// EAP paras
// Additional Services
EAP_paras^.AdditonalSerivce.Reserved1 := DINT_TO_REAL(EAP_para_DINT^.AdditonalSerivce.Reserved1);
EAP_paras^.AdditonalSerivce.Reserved2 := DINT_TO_REAL(EAP_para_DINT^.AdditonalSerivce.Reserved2);
EAP_paras^.AdditonalSerivce.Reserved3 := DINT_TO_REAL(EAP_para_DINT^.AdditonalSerivce.Reserved3);
EAP_paras^.AdditonalSerivce.Reserved4 := DINT_TO_REAL(EAP_para_DINT^.AdditonalSerivce.Reserved4);
EAP_paras^.AdditonalSerivce.Reserved5 := DINT_TO_REAL(EAP_para_DINT^.AdditonalSerivce.Reserved5);
EAP_paras^.AdditonalSerivce.Reserved6 := DINT_TO_REAL(EAP_para_DINT^.AdditonalSerivce.Reserved6);
EAP_paras^.AdditonalSerivce.Reserved7 := DINT_TO_REAL(EAP_para_DINT^.AdditonalSerivce.Reserved7);
EAP_paras^.AdditonalSerivce.Reserved8 := DINT_TO_REAL(EAP_para_DINT^.AdditonalSerivce.Reserved8);
EAP_paras^.AdditonalSerivce.Reserved9 := DINT_TO_REAL(EAP_para_DINT^.AdditonalSerivce.Reserved9);
EAP_paras^.AdditonalSerivce.Reserved10 := DINT_TO_REAL(EAP_para_DINT^.AdditonalSerivce.Reserved10);
EAP_paras^.AdditonalSerivce.Reserved11 := DINT_TO_REAL(EAP_para_DINT^.AdditonalSerivce.Reserved11);
EAP_paras^.AdditonalSerivce.Reserved12 := DINT_TO_REAL(EAP_para_DINT^.AdditonalSerivce.Reserved12);
EAP_paras^.AdditonalSerivce.Reserved13 := DINT_TO_REAL(EAP_para_DINT^.AdditonalSerivce.Reserved13);
EAP_paras^.AdditonalSerivce.Reserved14 := DINT_TO_REAL(EAP_para_DINT^.AdditonalSerivce.Reserved14);
EAP_paras^.AdditonalSerivce.Reserved15 := DINT_TO_REAL(EAP_para_DINT^.AdditonalSerivce.Reserved15);
EAP_paras^.AdditonalSerivce.Reserved16 := DINT_TO_REAL(EAP_para_DINT^.AdditonalSerivce.Reserved16);
//CommonBlock_Params
EAP_paras^.CommonBlock_Params_EAP.ActivePowerLimit := DINT_TO_REAL(EAP_para_DINT^.CommonBlock_Params_EAP.ActivePowerLimit);
EAP_paras^.CommonBlock_Params_EAP.Delta_limits := DINT_TO_REAL(EAP_para_DINT^.CommonBlock_Params_EAP.Delta_limits);
EAP_paras^.CommonBlock_Params_EAP.E_Limits := DINT_TO_REAL(EAP_para_DINT^.CommonBlock_Params_EAP.E_Limits)*0.1;
EAP_paras^.CommonBlock_Params_EAP.Ki_ReactiveControl := DINT_TO_REAL(EAP_para_DINT^.CommonBlock_Params_EAP.Ki_ReactiveControl)*0.0001;
EAP_paras^.CommonBlock_Params_EAP.Kp_ReactiveControl := DINT_TO_REAL(EAP_para_DINT^.CommonBlock_Params_EAP.Kp_ReactiveControl)*0.0001;
EAP_paras^.CommonBlock_Params_EAP.NominalFreq := DINT_TO_REAL(EAP_para_DINT^.CommonBlock_Params_EAP.NominalFreq);
EAP_paras^.CommonBlock_Params_EAP.NominalPower := DINT_TO_REAL(EAP_para_DINT^.CommonBlock_Params_EAP.NominalPower);
EAP_paras^.CommonBlock_Params_EAP.NominalVolt := DINT_TO_REAL(EAP_para_DINT^.CommonBlock_Params_EAP.NominalVolt);
EAP_paras^.CommonBlock_Params_EAP.ReactivePowerLimit := DINT_TO_REAL(EAP_para_DINT^.CommonBlock_Params_EAP.ReactivePowerLimit);
EAP_paras^.CommonBlock_Params_EAP.VirtualReactance := DINT_TO_REAL(EAP_para_DINT^.CommonBlock_Params_EAP.VirtualReactance)*0.001;
EAP_paras^.CommonBlock_Params_EAP.VirtualResistor := DINT_TO_REAL(EAP_para_DINT^.CommonBlock_Params_EAP.VirtualResistor)*0.001;
EAP_paras^.CommonBlock_Params_EAP.Reserved1 := DINT_TO_REAL(EAP_para_DINT^.CommonBlock_Params_EAP.Reserved1);
EAP_paras^.CommonBlock_Params_EAP.Reserved2 := DINT_TO_REAL(EAP_para_DINT^.CommonBlock_Params_EAP.Reserved2);
EAP_paras^.CommonBlock_Params_EAP.Reserved3 := DINT_TO_REAL(EAP_para_DINT^.CommonBlock_Params_EAP.Reserved3);
EAP_paras^.CommonBlock_Params_EAP.Reserved4 := DINT_TO_REAL(EAP_para_DINT^.CommonBlock_Params_EAP.Reserved4);
EAP_paras^.CommonBlock_Params_EAP.Reserved5 := DINT_TO_REAL(EAP_para_DINT^.CommonBlock_Params_EAP.Reserved5);
//FrequencyRegulation_Params
EAP_paras^.FrequencyRegulation_Params_EAP.DeadBand_Limits_P := DINT_TO_REAL(EAP_para_DINT^.FrequencyRegulation_Params_EAP.DeadBand_Limits_P)*0.1;
EAP_paras^.FrequencyRegulation_Params_EAP.DroopConstantP := DINT_TO_REAL(EAP_para_DINT^.FrequencyRegulation_Params_EAP.DroopConstantP)*0.1;
EAP_paras^.FrequencyRegulation_Params_EAP.LowPassFilter_CutOff_Freq := DINT_TO_REAL(EAP_para_DINT^.FrequencyRegulation_Params_EAP.LowPassFilter_CutOff_Freq)*0.01;
EAP_paras^.FrequencyRegulation_Params_EAP.Max_Delta_Energy := DINT_TO_REAL(EAP_para_DINT^.FrequencyRegulation_Params_EAP.Max_Delta_Energy);
EAP_paras^.FrequencyRegulation_Params_EAP.PowerLimit_Freq := DINT_TO_REAL(EAP_para_DINT^.FrequencyRegulation_Params_EAP.PowerLimit_Freq);
EAP_paras^.FrequencyRegulation_Params_EAP.Reserved1 := DINT_TO_REAL(EAP_para_DINT^.FrequencyRegulation_Params_EAP.Reserved1);
EAP_paras^.FrequencyRegulation_Params_EAP.Reserved2 := DINT_TO_REAL(EAP_para_DINT^.FrequencyRegulation_Params_EAP.Reserved2);
EAP_paras^.FrequencyRegulation_Params_EAP.Reserved3 := DINT_TO_REAL(EAP_para_DINT^.FrequencyRegulation_Params_EAP.Reserved3);
EAP_paras^.FrequencyRegulation_Params_EAP.Reserved4 := DINT_TO_REAL(EAP_para_DINT^.FrequencyRegulation_Params_EAP.Reserved4);
EAP_paras^.FrequencyRegulation_Params_EAP.Reserved5 := DINT_TO_REAL(EAP_para_DINT^.FrequencyRegulation_Params_EAP.Reserved5);
EAP_paras^.FrequencyRegulation_Params_EAP.Reserved6 := DINT_TO_REAL(EAP_para_DINT^.FrequencyRegulation_Params_EAP.Reserved6);
EAP_paras^.FrequencyRegulation_Params_EAP.Reserved7 := DINT_TO_REAL(EAP_para_DINT^.FrequencyRegulation_Params_EAP.Reserved7);
EAP_paras^.FrequencyRegulation_Params_EAP.Reserved8 := DINT_TO_REAL(EAP_para_DINT^.FrequencyRegulation_Params_EAP.Reserved8);
EAP_paras^.FrequencyRegulation_Params_EAP.Reserved9 := DINT_TO_REAL(EAP_para_DINT^.FrequencyRegulation_Params_EAP.Reserved9);
EAP_paras^.FrequencyRegulation_Params_EAP.Reserved10 := DINT_TO_REAL(EAP_para_DINT^.FrequencyRegulation_Params_EAP.Reserved10);
EAP_paras^.FrequencyRegulation_Params_EAP.Reserved11 := DINT_TO_REAL(EAP_para_DINT^.FrequencyRegulation_Params_EAP.Reserved11);
//InertiaEmulation_Params
EAP_paras^.InertiaEmulation_Params_EAP.Damping_Constant := DINT_TO_REAL(EAP_para_DINT^.InertiaEmulation_Params_EAP.Damping_Constant)*0.1;
EAP_paras^.InertiaEmulation_Params_EAP.HighPassFilterConst := DINT_TO_REAL(EAP_para_DINT^.InertiaEmulation_Params_EAP.HighPassFilterConst)*0.001;
EAP_paras^.InertiaEmulation_Params_EAP.Inertia_Constant := DINT_TO_REAL(EAP_para_DINT^.InertiaEmulation_Params_EAP.Inertia_Constant)*0.1;
EAP_paras^.InertiaEmulation_Params_EAP.Max_ROCOF := DINT_TO_REAL(EAP_para_DINT^.InertiaEmulation_Params_EAP.Max_ROCOF)*0.01;
EAP_paras^.InertiaEmulation_Params_EAP.Reserved1 := DINT_TO_REAL(EAP_para_DINT^.InertiaEmulation_Params_EAP.Reserved1);
EAP_paras^.InertiaEmulation_Params_EAP.Reserved2 := DINT_TO_REAL(EAP_para_DINT^.InertiaEmulation_Params_EAP.Reserved2);
EAP_paras^.InertiaEmulation_Params_EAP.Reserved3 := DINT_TO_REAL(EAP_para_DINT^.InertiaEmulation_Params_EAP.Reserved3);
EAP_paras^.InertiaEmulation_Params_EAP.Reserved4 := DINT_TO_REAL(EAP_para_DINT^.InertiaEmulation_Params_EAP.Reserved4);
EAP_paras^.InertiaEmulation_Params_EAP.Reserved5 := DINT_TO_REAL(EAP_para_DINT^.InertiaEmulation_Params_EAP.Reserved5);
EAP_paras^.InertiaEmulation_Params_EAP.Reserved6 := DINT_TO_REAL(EAP_para_DINT^.InertiaEmulation_Params_EAP.Reserved6);
EAP_paras^.InertiaEmulation_Params_EAP.Reserved7 := DINT_TO_REAL(EAP_para_DINT^.InertiaEmulation_Params_EAP.Reserved7);
EAP_paras^.InertiaEmulation_Params_EAP.Reserved8 := DINT_TO_REAL(EAP_para_DINT^.InertiaEmulation_Params_EAP.Reserved8);
EAP_paras^.InertiaEmulation_Params_EAP.Reserved9 := DINT_TO_REAL(EAP_para_DINT^.InertiaEmulation_Params_EAP.Reserved9);
EAP_paras^.InertiaEmulation_Params_EAP.Reserved10 := DINT_TO_REAL(EAP_para_DINT^.InertiaEmulation_Params_EAP.Reserved10);
EAP_paras^.InertiaEmulation_Params_EAP.Reserved11 := DINT_TO_REAL(EAP_para_DINT^.InertiaEmulation_Params_EAP.Reserved11);
EAP_paras^.InertiaEmulation_Params_EAP.Reserved12 := DINT_TO_REAL(EAP_para_DINT^.InertiaEmulation_Params_EAP.Reserved12);
//ModalFrequency_Params_EAP
EAP_paras^.ModalFrequency_Params_EAP.BandPassFilter_CenterFreq := DINT_TO_REAL(EAP_para_DINT^.ModalFrequency_Params_EAP.BandPassFilter_CenterFreq)*0.01;
EAP_paras^.ModalFrequency_Params_EAP.Max_ROCOF_Modal := DINT_TO_REAL(EAP_para_DINT^.ModalFrequency_Params_EAP.Max_ROCOF_Modal)*0.1;
EAP_paras^.ModalFrequency_Params_EAP.ModalFreq_Gain := DINT_TO_REAL(EAP_para_DINT^.ModalFrequency_Params_EAP.ModalFreq_Gain)*0.1;
EAP_paras^.ModalFrequency_Params_EAP.ModalFreq_PowerLimit := DINT_TO_REAL(EAP_para_DINT^.ModalFrequency_Params_EAP.ModalFreq_PowerLimit);
EAP_paras^.ModalFrequency_Params_EAP.Reserved1 := DINT_TO_REAL(EAP_para_DINT^.ModalFrequency_Params_EAP.Reserved1);
EAP_paras^.ModalFrequency_Params_EAP.Reserved2 := DINT_TO_REAL(EAP_para_DINT^.ModalFrequency_Params_EAP.Reserved2);
EAP_paras^.ModalFrequency_Params_EAP.Reserved3 := DINT_TO_REAL(EAP_para_DINT^.ModalFrequency_Params_EAP.Reserved3);
EAP_paras^.ModalFrequency_Params_EAP.Reserved4 := DINT_TO_REAL(EAP_para_DINT^.ModalFrequency_Params_EAP.Reserved4);
EAP_paras^.ModalFrequency_Params_EAP.Reserved5 := DINT_TO_REAL(EAP_para_DINT^.ModalFrequency_Params_EAP.Reserved5);
EAP_paras^.ModalFrequency_Params_EAP.Reserved6 := DINT_TO_REAL(EAP_para_DINT^.ModalFrequency_Params_EAP.Reserved6);
EAP_paras^.ModalFrequency_Params_EAP.Reserved7 := DINT_TO_REAL(EAP_para_DINT^.ModalFrequency_Params_EAP.Reserved7);
EAP_paras^.ModalFrequency_Params_EAP.Reserved8 := DINT_TO_REAL(EAP_para_DINT^.ModalFrequency_Params_EAP.Reserved8);
EAP_paras^.ModalFrequency_Params_EAP.Reserved9 := DINT_TO_REAL(EAP_para_DINT^.ModalFrequency_Params_EAP.Reserved9);
EAP_paras^.ModalFrequency_Params_EAP.Reserved10 := DINT_TO_REAL(EAP_para_DINT^.ModalFrequency_Params_EAP.Reserved10);
EAP_paras^.ModalFrequency_Params_EAP.Reserved11 := DINT_TO_REAL(EAP_para_DINT^.ModalFrequency_Params_EAP.Reserved11);
EAP_paras^.ModalFrequency_Params_EAP.Reserved12 := DINT_TO_REAL(EAP_para_DINT^.ModalFrequency_Params_EAP.Reserved12);
//VoltageRegulation_Params
EAP_paras^.VoltageRegulation_Params_EAP.DeadBand_Limit_Q := DINT_TO_REAL(EAP_para_DINT^.VoltageRegulation_Params_EAP.DeadBand_Limit_Q)*0.1;
EAP_paras^.VoltageRegulation_Params_EAP.DroopConstantQ := DINT_TO_REAL(EAP_para_DINT^.VoltageRegulation_Params_EAP.DroopConstantQ)*0.1;
EAP_paras^.VoltageRegulation_Params_EAP.LowPassFilter_CutOff_Volt := DINT_TO_REAL(EAP_para_DINT^.VoltageRegulation_Params_EAP.LowPassFilter_CutOff_Volt)*0.01;
EAP_paras^.VoltageRegulation_Params_EAP.PowerLimit_Volt := DINT_TO_REAL(EAP_para_DINT^.VoltageRegulation_Params_EAP.PowerLimit_Volt);
EAP_paras^.VoltageRegulation_Params_EAP.Reserved1 := DINT_TO_REAL(Modbus_para_DINT^.VoltageRegulation_Params.Reserved1);
EAP_paras^.VoltageRegulation_Params_EAP.Reserved2 := DINT_TO_REAL(Modbus_para_DINT^.VoltageRegulation_Params.Reserved2);
EAP_paras^.VoltageRegulation_Params_EAP.Reserved3 := DINT_TO_REAL(Modbus_para_DINT^.VoltageRegulation_Params.Reserved3);
EAP_paras^.VoltageRegulation_Params_EAP.Reserved4 := DINT_TO_REAL(Modbus_para_DINT^.VoltageRegulation_Params.Reserved4);
EAP_paras^.VoltageRegulation_Params_EAP.Reserved5 := DINT_TO_REAL(Modbus_para_DINT^.VoltageRegulation_Params.Reserved5);
EAP_paras^.VoltageRegulation_Params_EAP.Reserved6 := DINT_TO_REAL(Modbus_para_DINT^.VoltageRegulation_Params.Reserved6);
EAP_paras^.VoltageRegulation_Params_EAP.Reserved7 := DINT_TO_REAL(Modbus_para_DINT^.VoltageRegulation_Params.Reserved7);
EAP_paras^.VoltageRegulation_Params_EAP.Reserved8 := DINT_TO_REAL(Modbus_para_DINT^.VoltageRegulation_Params.Reserved8);
EAP_paras^.VoltageRegulation_Params_EAP.Reserved9 := DINT_TO_REAL(Modbus_para_DINT^.VoltageRegulation_Params.Reserved9);
EAP_paras^.VoltageRegulation_Params_EAP.Reserved10 := DINT_TO_REAL(Modbus_para_DINT^.VoltageRegulation_Params.Reserved10);
EAP_paras^.VoltageRegulation_Params_EAP.Reserved11 := DINT_TO_REAL(Modbus_para_DINT^.VoltageRegulation_Params.Reserved11);
EAP_paras^.VoltageRegulation_Params_EAP.Reserved12 := DINT_TO_REAL(Modbus_para_DINT^.VoltageRegulation_Params.Reserved12);

// EtherCAT inputs
EtherCAT_inputs^.ActivePowerReference := DINT_TO_REAL(EtherCAT_input_DINT^.ActivePowerReference);
EtherCAT_inputs^.Command := (EtherCAT_input_DINT^.Command);
EtherCAT_inputs^.Heartbeat := DINT_TO_REAL(EtherCAT_input_DINT^.Heartbeat);
EtherCAT_inputs^.ReactivePowerReference := DINT_TO_REAL(EtherCAT_input_DINT^.ReactivePowerReference);
EtherCAT_inputs^.Reserved4 := DINT_TO_REAL(EtherCAT_input_DINT^.Reserved4);
EtherCAT_inputs^.Reserved5 := DINT_TO_REAL(EtherCAT_input_DINT^.Reserved4);
EtherCAT_inputs^.Reserved6 := DINT_TO_REAL(EtherCAT_input_DINT^.Reserved4);
EtherCAT_inputs^.Reserved7 := DINT_TO_REAL(EtherCAT_input_DINT^.Reserved4);
EtherCAT_inputs^.Reserved8 := DINT_TO_REAL(EtherCAT_input_DINT^.Reserved4);
EtherCAT_inputs^.Reserved9 := DINT_TO_REAL(EtherCAT_input_DINT^.Reserved4);
EtherCAT_inputs^.Reserved10 := DINT_TO_REAL(EtherCAT_input_DINT^.Reserved4);
EtherCAT_inputs^.Reserved11 := DINT_TO_REAL(EtherCAT_input_DINT^.Reserved4);
EtherCAT_inputs^.Reserved12 := DINT_TO_REAL(EtherCAT_input_DINT^.Reserved4);
EtherCAT_inputs^.Reserved13 := DINT_TO_REAL(EtherCAT_input_DINT^.Reserved4);
EtherCAT_inputs^.Reserved14 := DINT_TO_REAL(EtherCAT_input_DINT^.Reserved4);
EtherCAT_inputs^.Reserved15 := DINT_TO_REAL(EtherCAT_input_DINT^.Reserved4);

// Monitoring information
EtherCAT_monitor_DINT^.BatSoc := REAL_TO_DINT(EtherCAT_monitor_var^.BatSoc*100);
EtherCAT_monitor_DINT^.BatSocLowLim := REAL_TO_DINT(EtherCAT_monitor_var^.BatSocLowLim*100);
EtherCAT_monitor_DINT^.BatSocUpLim := REAL_TO_DINT(EtherCAT_monitor_var^.BatSocUpLim*100);
EtherCAT_monitor_DINT^.GridFre := REAL_TO_DINT(EtherCAT_monitor_var^.GridFre*100);
EtherCAT_monitor_DINT^.Irmsa := REAL_TO_DINT(EtherCAT_monitor_var^.Irmsa*100);
EtherCAT_monitor_DINT^.Irmsb := REAL_TO_DINT(EtherCAT_monitor_var^.Irmsb*100);
EtherCAT_monitor_DINT^.Irmsc := REAL_TO_DINT(EtherCAT_monitor_var^.Irmsc*100);
EtherCAT_monitor_DINT^.MaxVArAval := REAL_TO_DINT(EtherCAT_monitor_var^.MaxVArAval*100);
EtherCAT_monitor_DINT^.MaxWAval := REAL_TO_DINT(EtherCAT_monitor_var^.MaxWAval*100);
EtherCAT_monitor_DINT^.MaxWCharVal := REAL_TO_DINT(EtherCAT_monitor_var^.MaxWCharVal*100);
EtherCAT_monitor_DINT^.MinVArAval := REAL_TO_DINT(EtherCAT_monitor_var^.MinVArAval*100);
EtherCAT_monitor_DINT^.TotVAr := REAL_TO_DINT(EtherCAT_monitor_var^.TotVAr);
EtherCAT_monitor_DINT^.TotW := REAL_TO_DINT(EtherCAT_monitor_var^.TotW);
EtherCAT_monitor_DINT^.Vrmsa := REAL_TO_DINT(EtherCAT_monitor_var^.Vrmsa*100);
EtherCAT_monitor_DINT^.Vrmsb := REAL_TO_DINT(EtherCAT_monitor_var^.Vrmsb*100);
EtherCAT_monitor_DINT^.Vrmsc := REAL_TO_DINT(EtherCAT_monitor_var^.Vrmsc*100);

END_FUNCTION

// ---- Functions/Communications/Mapping_Monitoring_Variables.TcPOU
FUNCTION Mapping_Monitoring_Variables
VAR_INPUT
	Input_var : ScaledModRead;
	Output_var : POINTER TO EtherCAT_Monitor_Variables;
	Output_var2 : POINTER TO EtherCAT_Stat_Variables;
END_VAR
VAR
END_VAR

Output_var^.BatSoc := Input_var.BatSoc;
Output_var^.BatSocLowLim := Input_var.BatSocLowLimit;
Output_var^.BatSocUpLim := Input_var.BatSocUpLimit;

Output_var2^.Status := Input_var.fbOpMode;
Output_var2^.HeartBeat := GlobalVar.wMiliseconds;

Output_var2^.Alarms1 := Input_var.GrAlm0;
Output_var2^.Alarms2 := Input_var.GrAlm1;
Output_var2^.Alarms3 := Input_var.GrAlm2;
Output_var2^.Alarms4 := Input_var.GrAlm3;

Output_var^.GridFre := Input_var.GridFre;

Output_var^.Irmsa := Input_var.Irmsa;
Output_var^.Irmsb := Input_var.Irmsb;
Output_var^.Irmsc := Input_var.Irmsc;

Output_var^.TotW := Input_var.TotW;
Output_var^.TotVAr := Input_var.TotVAr;

Output_var^.Vrmsa := Input_var.Vrmsa;
Output_var^.Vrmsb := Input_var.Vrmsb;
Output_var^.Vrmsc := Input_var.Vrmsc;

END_FUNCTION

// ---- Functions/Communications/Mapping_Monitoring_Variables_ABG.TcPOU
FUNCTION Mapping_Monitoring_Variables_ABG
VAR_INPUT
	Input_var : ModbusRead;//ScaledModRead;
	Output_var : POINTER TO EtherCAT_Monitor_Variables;
	Output_var2 : POINTER TO EtherCAT_Stat_Variables;
END_VAR
VAR
END_VAR

Output_var^.BatSoc := (Input_var.BatSoc );
Output_var^.BatSocLowLim := (Input_var.BatSocLowLim);
Output_var^.BatSocUpLim := (Input_var.BatSocUpLim );

CASE Input_var.DerOpMode	OF
	0:	
		Output_var2^.Status := 0;
	1:	
		Output_var2^.Status := 0;
	4:
		Output_var2^.Status := 1;
	11:
		Output_var2^.Status := 1;
	5:
		Output_var2^.Status := 2;
	6:
		Output_var2^.Status := 3;
	9:
		Output_var2^.Status := 5;
END_CASE

//Output_var2^.Status := Input_var.DerOpMode;


Output_var2^.HeartBeat := GlobalVar.wMiliseconds;

Output_var2^.Alarms1 := UDINT_TO_DINT((Input_var.GrAlm));
Output_var2^.Alarms2 := 0; //Input_var.GrAlm1;
Output_var2^.Alarms3 := 0; //Input_var.GrAlm2;
Output_var2^.Alarms4 := 0; //Input_var.GrAlm3;

Output_var^.GridFre := (Input_var.GridFre);

Output_var^.Irmsa := (Input_var.Irmsa);
Output_var^.Irmsb := (Input_var.Irmsb);
Output_var^.Irmsc := (Input_var.Irmsc);

Output_var^.TotW := (Input_var.TotW);
Output_var^.TotVAr := (Input_var.TotVAr);

Output_var^.Vrmsa := (Input_var.Vrmsa);
Output_var^.Vrmsb := (Input_var.Vrmsb);
Output_var^.Vrmsc := (Input_var.Vrmsc);

END_FUNCTION

// ---- Programs/Timer.TcPOU
PROGRAM Timer
VAR
	cnt	:	INT;
END_VAR

//Timer 1 ms
	GlobalVar.wMiliseconds := GlobalVar.wMiliseconds +1;
	IF GlobalVar.wMiliseconds >1000 THEN 
		GlobalVar.wMiliseconds := 0;
	END_IF

// Event Recorder
// Transmiting part of historian
cnt := cnt + 1;
IF cnt = 50 THEN
	cnt := 0;
	gvl.fbHistorian.Transmiting(HistorianDataPacket_EtherCAT => gvl.HistorianDataPacket_EtherCAT);		
	gvl.HistorianDataPacket_EtherCAT.TransmitRequest := gvl.fbHistorian.GetRequest;

END_IF

END_PROGRAM

// ---- Functions/EventRecoder/UnixTimestamp.TcPOU
FUNCTION_BLOCK UnixTimestamp
VAR_OUTPUT
    seconds: ULINT;
    milliseconds: ULINT;
END_VAR

VAR
    localSystemTime : FB_LocalSystemTime := ( bEnable := TRUE, dwCycle := 1 );
    getTimeZoneInformation : FB_GetTimeZoneInformation;
    timeZoneInformation : ST_TimeZoneInformation;
    specificLocalTimeToFileTime : FB_TzSpecificLocalTimeToFileTime;
    fileTime: T_FILETIME;
    onZerothSecondLastCycle : BOOL;
END_VAR

// Get local system time
localSystemTime();

// On the zeroth second of each minutesync timezone information
IF (timeZoneInformation.standardName = '' OR (localSystemTime.systemTime.wSecond = 0 AND NOT onZerothSecondLastCycle)) THEN
    getTimeZoneInformation(sNetID := '', bExecute := TRUE, tzInfo => timeZoneInformation);
END_IF;

// Convert local system time to unix timestamps
specificLocalTimeToFileTime(in := Tc2_Utilities.SYSTEMTIME_TO_FILETIME(localSystemTime.systemTime), tzInfo := timeZoneInformation, out => fileTime);
seconds := (SHL(DWORD_TO_ULINT(fileTime.dwHighDateTime), 32) + DWORD_TO_ULINT(fileTime.dwLowDateTime)) / 10000000 - 11644473600;
milliseconds := (SHL(DWORD_TO_ULINT(fileTime.dwHighDateTime), 32) + DWORD_TO_ULINT(fileTime.dwLowDateTime)) / 10000 - 11644473600000;

onZerothSecondLastCycle := localSystemTime.systemTime.wSecond = 0;

END_FUNCTION_BLOCK

// ---- Functions/EventRecoder/HistorianFunctionBlock.TcPOU
FUNCTION_BLOCK HistorianFunctionBlock
VAR_INPUT
	
END_VAR

VAR_OUTPUT
	
END_VAR

VAR
	HistorianStateMachine			:	UINT	:=	3;
	
	FIFO_Buffer_In_Modbus			:	ARRAY [0..1199] OF EventRecorder_In_Modbus;
	FIFO_Buffer_In_EAP 				:	ARRAY [0..1199] OF EventRecorder_In_EAP;
	FIFO_Buffer_ControllerOut 		:	ARRAY [0..1199] OF EventRecorder_Controller_Output;
	FIFO_Buffer_Index_TimeStamp		:	ARRAY [0..1199] OF Index_TimeStamp;	
	
	
	FIFO_Transmit_EAP_Index			:	INT;
	FIFO_Transmit_Modbus_Index		:	INT;
	FIFO_Transmit_ControlOut_Index	:	INT;
	
	
	FIFO_Index_Max					:	INT := 1200;
	PreEventCaptures				:	INT	:= 200;	// 20 Percent of preevent recored
	
	FIFO_StopIndex					:	INT;
	FIFO_StopIndex_Modbus			:	INT;
	FIFO_StopIndex_ControlOut		:	INT;
	
	FIFO_index						:	INT;
	FIFO_index_Modbus				:	INT;
	FIFO_index_ControlOut			:	INT;
	
	
	TranmitingIndex					:	INT;
	RecordingTriger					:	BOOL;
	_TransmitRequest				:	INT;
	FIFO_Transmit_Index				:	INT;
	
	EAP_Record_done			:	BOOL := FALSE;
	Modbus_Record_done		:	BOOL := FALSE;
	ControlOut_Record_done	:	BOOL := FALSE;
	
	EAP_trigger_done		:	BOOL := FALSE;
	Modbus_triger_done		:	BOOL := FALSE;
	ControlOut_triger_done	:	BOOL := FALSE;
		
	unixTime: UnixTimestamp;
    timestampSeconds: ULINT;
    timestampMilliseconds: ULINT;
	

END_VAR

PROPERTY GetRequest : INT;
GET
GetRequest	:=	_TransmitRequest;
END_GET
END_PROPERTY

METHOD PUBLIC ListeningRecording_ControlOut : BOOL
VAR_INPUT
	HistorianDataPacket		:	EventRecorder_Controller_Output;
END_VAR

VAR_OUTPUT
	
END_VAR

VAR
	icounter	:	INT;
END_VAR
// State machine for Historian
IF EAP_trigger_done AND NOT ControlOut_triger_done AND RecordingTriger THEN
	// Set stop index with buffer wrapping
		FIFO_StopIndex_ControlOut := FIFO_index_ControlOut - PreEventCaptures;	//	Set the end of FIFO buffer
		IF FIFO_StopIndex_ControlOut < 0 THEN							// wrapping
			FIFO_StopIndex_ControlOut := FIFO_Index_Max + FIFO_StopIndex_ControlOut;
		END_IF
		// Go to the recording State
		HistorianStateMachine := 1;
		ControlOut_triger_done := TRUE;
END_IF
CASE HistorianStateMachine	OF
//---------------- Begin of Listening State -------------------------------	
	0:	// Listening
		FIFO_index_ControlOut := FIFO_index_ControlOut + 1;							// Inceasing buffer index
		IF FIFO_index_ControlOut = FIFO_Index_Max THEN						// Buffer wrapping
			FIFO_index_ControlOut := 0;
		END_IF	
	
		FIFO_Buffer_ControllerOut[FIFO_index_ControlOut] := HistorianDataPacket;			// Copy data to buffer
		
		IF RecordingTriger = TRUE AND NOT ControlOut_triger_done THEN
			// Set stop index with buffer wrapping
			FIFO_StopIndex_ControlOut := FIFO_index_ControlOut - PreEventCaptures;	//	Set the end of FIFO buffer
			IF FIFO_StopIndex_ControlOut < 0 THEN							// wrapping
				FIFO_StopIndex_ControlOut := FIFO_Index_Max + FIFO_StopIndex_ControlOut;
			END_IF
			// Go to the recording State
			HistorianStateMachine := 1;
		END_IF
//---------------- End of Listening State   -------------------------------	

//---------------- Begin of Recording State -------------------------------		
	1:	
		IF NOT ControlOut_Record_done THEN
	
			FIFO_index_ControlOut := FIFO_index_ControlOut + 1;					// Inceasing buffer index
			IF FIFO_index_ControlOut = FIFO_Index_Max THEN				// Buffer wrapping
				FIFO_index_ControlOut := 0;
			END_IF
			
			FIFO_Buffer_ControllerOut[FIFO_index_ControlOut] := HistorianDataPacket;	
			
			IF FIFO_index_ControlOut = FIFO_StopIndex_ControlOut THEN				// change to transmit state
				ControlOut_Record_done	:= TRUE;					// Send request
			END_IF
		END_IF
		
	3: // Initialization
		FOR icounter :=	0 TO (FIFO_Index_Max-1)	BY 1 DO
			FIFO_Buffer_Index_Timestamp[icounter].Index := icounter;
		END_FOR
		HistorianStateMachine := 0;
END_CASE
END_METHOD

METHOD PUBLIC ListeningRecording_IN_EAP : BOOL
VAR_INPUT
	HistorianDataPacket		:	EventRecorder_In_EAP;
END_VAR

VAR_OUTPUT
	
END_VAR

VAR
	icounter	:	INT;
END_VAR
// State machine for Historian

CASE HistorianStateMachine	OF
//---------------- Begin of Listening State -------------------------------	
	0:	// Listening
		FIFO_index := FIFO_index + 1;							// Inceasing buffer index
		IF FIFO_index = FIFO_Index_Max THEN						// Buffer wrapping
			FIFO_index := 0;
		END_IF	
	
		FIFO_Buffer_In_EAP[FIFO_index] := HistorianDataPacket;			// Copy data to buffer
		
		IF RecordingTriger = TRUE AND NOT EAP_trigger_done THEN
			// Set stop index with buffer wrapping
			FIFO_StopIndex := FIFO_index - PreEventCaptures;	//	Set the end of FIFO buffer
			IF FIFO_StopIndex < 0 THEN							// wrapping
				FIFO_StopIndex := FIFO_Index_Max + FIFO_StopIndex;
			END_IF
			// Go to the recording State
			EAP_trigger_done := TRUE;
			HistorianStateMachine := 1;
		END_IF
//---------------- End of Listening State   -------------------------------	

//---------------- Begin of Recording State -------------------------------		
	1:	
		
		IF NOT EAP_Record_done THEN
	
			FIFO_index := FIFO_index + 1;					// Inceasing buffer index
			IF FIFO_index = FIFO_Index_Max THEN				// Buffer wrapping
				FIFO_index := 0;
			END_IF
			
			FIFO_Buffer_In_EAP[FIFO_index] := HistorianDataPacket;	
			
			IF FIFO_index = FIFO_StopIndex THEN				// change to transmit state
				EAP_Record_done	:= TRUE;					// Send request
			END_IF
		END_IF
		
	3: // Initialization
		FOR icounter :=	0 TO (FIFO_Index_Max-1)	BY 1 DO
			FIFO_Buffer_Index_Timestamp[icounter].Index := icounter;
		END_FOR
		HistorianStateMachine := 0;
END_CASE
END_METHOD

METHOD ListeningRecording_IN_Modbus : BOOL
VAR_INPUT
	HistorianDataPacket		:	EventRecorder_In_Modbus;
END_VAR

VAR_OUTPUT
	
END_VAR

VAR
	icounter	:	INT;
END_VAR
// Unix Time
Globalvar.unixTime();
Globalvar.timestampMilliseconds := ULINT_TO_UINT(Globalvar.unixTime.milliseconds - Globalvar.unixTime.seconds*1000);
Globalvar.timestampSeconds.dwSecond := ULINT_TO_DWORD(Globalvar.unixTime.seconds);


// State machine for Historian
IF EAP_trigger_done AND NOT Modbus_Triger_done AND RecordingTriger THEN
	// Set stop index with buffer wrapping
			FIFO_StopIndex_Modbus := FIFO_index_Modbus - PreEventCaptures;	//	Set the end of FIFO buffer
			IF FIFO_StopIndex_Modbus < 0 THEN								// wrapping
				FIFO_StopIndex_Modbus := FIFO_Index_Max + FIFO_StopIndex_Modbus;
			END_IF
			// Go to the recording State
			HistorianStateMachine := 1;
			Modbus_Triger_done := TRUE;
END_IF
CASE HistorianStateMachine	OF
//---------------- Begin of Listening State -------------------------------	
	0:	// Listening
		FIFO_index_Modbus := FIFO_index_Modbus + 1;							// Inceasing buffer index
		IF FIFO_index_Modbus = FIFO_Index_Max THEN						// Buffer wrapping
			FIFO_index_Modbus := 0;
		END_IF	
	
		FIFO_Buffer_In_Modbus[FIFO_index_Modbus] := HistorianDataPacket;			// Copy data to buffer
		FIFO_Buffer_Index_TimeStamp[FIFO_index_Modbus].TimeStamp := Globalvar.timestampSeconds.dtSecond;
		FIFO_Buffer_Index_TimeStamp[FIFO_index_Modbus].Miliseconds := Globalvar.timestampMilliseconds;
		
		IF RecordingTriger = TRUE AND NOT Modbus_triger_done  THEN
			// Set stop index with buffer wrapping
			FIFO_StopIndex_Modbus := FIFO_index_Modbus - PreEventCaptures;	//	Set the end of FIFO buffer
			IF FIFO_StopIndex_Modbus < 0 THEN								// wrapping
				FIFO_StopIndex_Modbus := FIFO_Index_Max + FIFO_StopIndex_Modbus;
			END_IF
			// Go to the recording State
			HistorianStateMachine := 1;
		END_IF
//---------------- End of Listening State   -------------------------------	

//---------------- Begin of Recording State -------------------------------		
	1:	IF NOT 	Modbus_Record_done THEN
		
			FIFO_index_Modbus := FIFO_index_Modbus + 1;					// Inceasing buffer index
			IF FIFO_index_Modbus = FIFO_Index_Max THEN				// Buffer wrapping
				FIFO_index_Modbus := 0;
			END_IF
			
			FIFO_Buffer_In_Modbus[FIFO_index_Modbus] := HistorianDataPacket;	
			FIFO_Buffer_Index_TimeStamp[FIFO_index_Modbus].TimeStamp := Globalvar.timestampSeconds.dtSecond;
			FIFO_Buffer_Index_TimeStamp[FIFO_index_Modbus].Miliseconds := Globalvar.timestampMilliseconds;
			
			IF FIFO_index_Modbus = FIFO_StopIndex_Modbus THEN	// change to transmit state
				Modbus_Record_done := TRUE;						// Send request
			END_IF
		END_IF
END_CASE
END_METHOD

PROPERTY SetTtriger : BOOL
SET
RecordingTriger := SetTtriger;
END_SET
END_PROPERTY

METHOD PUBLIC Transmiting : BOOL
VAR_INPUT
	
END_VAR

VAR_OUTPUT
	HistorianDataPacket_EtherCAT	:	EthercatDataPacket;
END_VAR
IF EAP_Record_done AND Modbus_Record_done  AND ControlOut_Record_done THEN
	_TransmitRequest := 1;
	HistorianStateMachine := 2;
ELSE
	_TransmitRequest := 0;
END_IF

// State machine for Historian
CASE HistorianStateMachine	OF
//---------------- Begin of Transmiting State -----------------------------	
	2:
		IF gvl.TransmitApproved = 1  THEN
			
		// Increasing transmitting index
			FIFO_Transmit_Index := FIFO_Transmit_Index + 1;
		
			FIFO_Transmit_EAP_Index := FIFO_index + FIFO_Transmit_Index;
			FIFO_Transmit_Modbus_Index := FIFO_index_Modbus + FIFO_Transmit_Index;
			FIFO_Transmit_ControlOut_Index := FIFO_index_ControlOut + FIFO_Transmit_Index;
			
			IF FIFO_Transmit_EAP_Index >= FIFO_Index_Max THEN					// Buffer wrapping
				FIFO_Transmit_EAP_Index := FIFO_Transmit_EAP_Index - FIFO_Index_Max;
			END_IF
			
			IF FIFO_Transmit_Modbus_Index >= FIFO_Index_Max THEN					// Buffer wrapping
				FIFO_Transmit_Modbus_Index := FIFO_Transmit_Modbus_Index - FIFO_Index_Max;
			END_IF
			
			IF FIFO_Transmit_ControlOut_Index >= FIFO_Index_Max THEN					// Buffer wrapping
				FIFO_Transmit_ControlOut_Index := FIFO_Transmit_ControlOut_Index - FIFO_Index_Max;
			END_IF
			
			HistorianDataPacket_EtherCAT.SingalIn_Modbus := FIFO_Buffer_In_Modbus[FIFO_Transmit_Modbus_Index];		// Map to EtherCAT
			HistorianDataPacket_EtherCAT.SignalIn_EAP := FIFO_Buffer_In_EAP[FIFO_Transmit_EAP_Index];			// Map to EtherCAT
			HistorianDataPacket_EtherCAT.ControllerOut := FIFO_Buffer_ControllerOut[FIFO_Transmit_ControlOut_Index];
			HistorianDataPacket_EtherCAT.Index_TimeStamp.Index := FIFO_Transmit_Index - 1;
			
			HistorianDataPacket_EtherCAT.Index_TimeStamp.TimeStamp := FIFO_Buffer_Index_TimeStamp[FIFO_Transmit_Modbus_Index].TimeStamp ;
			HistorianDataPacket_EtherCAT.Index_TimeStamp.Miliseconds := FIFO_Buffer_Index_TimeStamp[FIFO_Transmit_Modbus_Index].Miliseconds;
			
			// Done and Switch to listening State
			IF FIFO_Transmit_Index >= FIFO_Index_Max THEN
				FIFO_Transmit_Index := 0;		// Remove request
				HistorianStateMachine := 0;
				
				FIFO_index := 0;
				FIFO_index_Modbus := 0;
				FIFO_index_ControlOut := 0;
				
				EAP_Record_done := FALSE;
				Modbus_Record_done	:=	FALSE;
				ControlOut_Record_done := FALSE;
				
				EAP_trigger_done := FALSE;
				Modbus_Triger_done := FALSE;
				ControlOut_triger_done := FALSE;
				
			END_IF			
		END_IF
//---------------- End of Transmiting State -------------------------------	
END_CASE
END_METHOD

END_FUNCTION_BLOCK

// ---- Functions/Communications/EtherCAT_MappingEAP.TcPOU
FUNCTION EtherCAT_MappingEAP
VAR_INPUT
	EAP_Controller : POINTER TO EAP_SPC;
END_VAR
VAR
END_VAR

//Commands
	//Common Block - Commands
		EAP_Controller^.ActivePowerLimitation := Communications.EtherCAT_EAP_Commands.CommonBlock_EAP.Bits.ActivePowerLimitation;
		EAP_Controller^.ReactivePowerLimitation := Communications.EtherCAT_EAP_Commands.CommonBlock_EAP.Bits.ReactivePowerLimitation;
		EAP_Controller^.Delta_Limitation := Communications.EtherCAT_EAP_Commands.CommonBlock_EAP.Bits.Delta_Limitation;
		EAP_Controller^.E_Limitation := Communications.EtherCAT_EAP_Commands.CommonBlock_EAP.Bits.E_Limitation;
		EAP_Controller^.SOC_Limitation := Communications.EtherCAT_EAP_Commands.CommonBlock_EAP.Bits.SOC_Limitation;
		EAP_Controller^.Reset_To_Default_Common := Communications.EtherCAT_EAP_Commands.CommonBlock_EAP.Bits.Reset_To_Default_Common;
	//Inertia Emulation - Commands
		EAP_Controller^.Enable_Inertia := Communications.EtherCAT_EAP_Commands.InertiaEmulation_EAP.Bits.Enable_Inertia;
		EAP_Controller^.Reset_States_Inertia := Communications.EtherCAT_EAP_Commands.InertiaEmulation_EAP.Bits.Reset_States_Inertia;
		EAP_Controller^. ROCOF_Limitation := Communications.EtherCAT_EAP_Commands.InertiaEmulation_EAP.Bits.ROCOF_Limitation;
		EAP_Controller^.Reset_To_Default_Inertia := Communications.EtherCAT_EAP_Commands.InertiaEmulation_EAP.Bits.Reset_To_Default_Inertia;
	//Frequency Regulation - Commands
		EAP_Controller^.Enable_DroopP := Communications.EtherCAT_EAP_Commands.FrequencyRegulation_EAP.Bits.Enable_DroopP;
		EAP_Controller^.Enable_DeadBandFreq := Communications.EtherCAT_EAP_Commands.FrequencyRegulation_EAP.Bits.Enable_DeadBandFreq;
		EAP_Controller^.Delta_Power_Limitation_Freq := Communications.EtherCAT_EAP_Commands.FrequencyRegulation_EAP.Bits.Delta_Power_Limitation_freq;
		EAP_Controller^.Delta_Energy_Limitation := Communications.EtherCAT_EAP_Commands.FrequencyRegulation_EAP.Bits.Delta_Energy_Limitation;
		EAP_Controller^.Reset_To_Default_Freq := Communications.EtherCAT_EAP_Commands.FrequencyRegulation_EAP.Bits.Reset_To_Default_Freq;
	//Modal Frequency Attenuation - Commands
		EAP_Controller^.Enable_ModalFreq := Communications.EtherCAT_EAP_Commands.ModalFreq_EAP.Bits.Enable_ModalFreq;
		EAP_Controller^.ModalFreq_PowerLimitation := Communications.EtherCAT_EAP_Commands.ModalFreq_EAP.Bits.ModalFreq_PowerLimitation;
		EAP_Controller^.ROCOF_Limitation_ModalFreq := Communications.EtherCAT_EAP_Commands.ModalFreq_EAP.Bits.ROCOF_Limitation_ModalFreq;
		EAP_Controller^.Reset_To_Default_ModalFreq := Communications.EtherCAT_EAP_Commands.ModalFreq_EAP.Bits.Reset_To_Default_ModalFreq;
	//Voltage Regulation - Commands
		EAP_Controller^.Enable_VoltageRegulation := Communications.EtherCAT_EAP_Commands.VoltageRegulation_EAP.Bits.Enable_VoltageRegulation;
		EAP_Controller^.Enable_DeadBandV := Communications.EtherCAT_EAP_Commands.VoltageRegulation_EAP.Bits.Enable_deadBandV;
		EAP_Controller^.Delta_Power_Limitation_VoltReg := Communications.EtherCAT_EAP_Commands.VoltageRegulation_EAP.Bits.Delta_Power_Limitation_VoltReg;
		EAP_Controller^.Reset_To_Default_VoltReg := Communications.EtherCAT_EAP_Commands.VoltageRegulation_EAP.Bits.Reset_To_Default_VoltReg;
//Parameters
	//Common Block - Parameters
		EAP_Controller^.NominalPower := Communications.EtherCAT_EAP_Parameters.CommonBlock_Params_EAP.NominalPower;
		EAP_Controller^.NominalFreq := Communications.EtherCAT_EAP_Parameters.CommonBlock_Params_EAP.NominalFreq;
		EAP_Controller^.NominalVolt := Communications.EtherCAT_EAP_Parameters.CommonBlock_Params_EAP.NominalVolt;
		EAP_Controller^.ActivePowerLimit := Communications.EtherCAT_EAP_Parameters.CommonBlock_Params_EAP.ActivePowerLimit;
		EAP_Controller^.ReactivePowerLimit := Communications.EtherCAT_EAP_Parameters.CommonBlock_Params_EAP.ReactivePowerLimit;
		EAP_Controller^.Delta_Limits := Communications.EtherCAT_EAP_Parameters.CommonBlock_Params_EAP.Delta_limits;
		EAP_Controller^.E_Limits := Communications.EtherCAT_EAP_Parameters.CommonBlock_Params_EAP.E_Limits;
		EAP_Controller^.Kp_ReactiveControl := Communications.EtherCAT_EAP_Parameters.CommonBlock_Params_EAP.Kp_ReactiveControl;
		EAP_Controller^.Ki_ReactiveControl := Communications.EtherCAT_EAP_Parameters.CommonBlock_Params_EAP.Ki_ReactiveControl;
		EAP_Controller^.VirtualReactance := Communications.EtherCAT_EAP_Parameters.CommonBlock_Params_EAP.VirtualReactance;
		EAP_Controller^.VirtualResistance := Communications.EtherCAT_EAP_Parameters.CommonBlock_Params_EAP.VirtualResistor;
	//Inertia Emulation - Parameters
		EAP_Controller^.Inertia_Constant := Communications.EtherCAT_EAP_Parameters.InertiaEmulation_Params_EAP.Inertia_Constant;
		EAP_Controller^.Damping_Constant := Communications.EtherCAT_EAP_Parameters.InertiaEmulation_Params_EAP.Damping_Constant;
		EAP_Controller^.HighPassFilterConst := Communications.EtherCAT_EAP_Parameters.InertiaEmulation_Params_EAP.HighPassFilterConst;
		EAP_Controller^.Max_ROCOF := Communications.EtherCAT_EAP_Parameters.InertiaEmulation_Params_EAP.Max_ROCOF;
	//Frequency Regulation - Parameters
		EAP_Controller^.DroopConstantP := Communications.EtherCAT_EAP_Parameters.FrequencyRegulation_Params_EAP.DroopConstantP;
		EAP_Controller^.Max_Delta_Energy := Communications.EtherCAT_EAP_Parameters.FrequencyRegulation_Params_EAP.Max_Delta_Energy;
		EAP_Controller^.PowerLimit_Freq := Communications.EtherCAT_EAP_Parameters.FrequencyRegulation_Params_EAP.PowerLimit_Freq;
		EAP_Controller^.LowPassFilter_CutOff_Freq := Communications.EtherCAT_EAP_Parameters.FrequencyRegulation_Params_EAP.LowPassFilter_CutOff_Freq;
		EAP_Controller^.DeadBand_Limits_P := Communications.EtherCAT_EAP_Parameters.FrequencyRegulation_Params_EAP.DeadBand_Limits_P;
	//Modal Frequency Attenunation -  Parameters
		EAP_Controller^.ModalFreq_Gain := Communications.EtherCAT_EAP_Parameters.ModalFrequency_Params_EAP.ModalFreq_Gain;
		EAP_Controller^.ModalFreq_PowerLimit := Communications.EtherCAT_EAP_Parameters.ModalFrequency_Params_EAP.ModalFreq_PowerLimit;
		EAP_Controller^.Max_ROCOF_Modal := Communications.EtherCAT_EAP_Parameters.ModalFrequency_Params_EAP.Max_ROCOF_Modal;
		EAP_Controller^.BandPassFilter_CenterFreq := Communications.EtherCAT_EAP_Parameters.ModalFrequency_Params_EAP.BandPassFilter_CenterFreq;

END_FUNCTION

// ---- Functions/Filters/BandPassFilter.TcPOU
FUNCTION BandPassFilter : REAL
VAR_INPUT
	Error : REAL;
	
	BPF : POINTER TO BandPassFilterStruct;
	
	Enable : BOOL;
	
END_VAR
VAR
END_VAR

BandPassFilter := BPF^.G1_b0*(Error - BPF^.error2) - BPF^.output1*BPF^.G1_a1 - BPF^.output2*BPF^.G1_a2;

IF Enable = TRUE THEN
	BPF^.error1 := Error;
	BPF^.error2 := BPF^.error1;
	BPF^.output1 := BandPassFilter;
	BPF^.output2 := BPF^.output1;
ELSE
	BPF^.error1 := 0;
	BPF^.error2 := 0;
	BPF^.output1 := 0;
	BPF^.output2 := 0;
	BandPassFilter := 0;
END_IF

END_FUNCTION

// ---- Functions/Filters/BandPassFilterParameters.TcPOU
FUNCTION BandPassFilterParameters
VAR_INPUT
	Damping : REAL;
	WCentral : REAL;
	
	BPF : POINTER TO BandPassFilterStruct;
	
	TS : REAL;
END_VAR
VAR
	WBase_2 : REAL;
	Q: REAL;
END_VAR

WBase_2 := WCentral*WCentral;
Q := 1 / (2 * Damping);

//Denominator G1
BPF^.G1_a0 := 1 / (TS*TS*WBASE_2*Q + 2 * WCentral*TS + 4 * Q);
BPF^.G1_a1 := BPF^.G1_a0*(2 * WBase_2*TS*TS*Q - 8 * Q);
BPF^.G1_a2 := BPF^.G1_a0*(TS*TS*WBase_2*Q - 2 * WCentral*TS + 4 * Q);
//Numerator
BPF^.G1_b0 := BPF^.G1_a0*(2 * WCentral*TS);

END_FUNCTION

// ---- Functions/Filters/LPF_FilterInit.TcPOU
FUNCTION LPF_FilterInit
VAR_INPUT
	CutFreq : REAL;
	Filter : POINTER TO LowPassFilter;
	TS : REAL;
END_VAR
VAR
END_VAR

Filter^.FrequencyCut := CutFreq;
Filter^.CutFreq := 1/1/(2*3.1415*Filter^.FrequencyCut);


Filter^.Den := 1/(TS + 2*(Filter^.CutFreq));
	
Filter^.a1 := (TS - 2*Filter^.CutFreq)*Filter^.Den;
Filter^.b0 := TS*Filter^.Den;
Filter^.b1 := TS*Filter^.Den;

END_FUNCTION

// ---- Functions/Filters/LPF_Function.TcPOU
FUNCTION LPF_Function : REAL
VAR_INPUT
	SignalToFilter : REAL;
	FilterParams : POINTER TO LowPassFilter;
END_VAR
VAR
END_VAR

LPF_Function := FilterParams^.b0*SignalToFilter + FilterParams^.b1*FilterParams^.ErrorFilt - FilterParams^.OutputFilt*FilterParams^.a1;
FilterParams^.ErrorFilt := SignalToFilter;
FilterParams^.OutputFilt := LPF_Function;

END_FUNCTION
